// TIA Portal V17 export
// export: Created 2026-05-13T16:54:41.7855142Z, ExportSetting WithDefaults, DisplayName Totally Integrated Automation Portal, DisplayVersion V17 Update 4, DisplayName TIA Portal Openness, DisplayVersion V17 Update 4, DisplayName TIA Portal Version Control Interface, DisplayVersion V17, DisplayName SINAMICS Startdrive Advanced, DisplayVersion V17, DisplayName SINAMICS Startdrive G130, G150, S120, S150, SINAMICS MV, S210, DisplayVersion V17, DisplayName SINAMICS Startdrive G110M, G120, G120C, G120D, G120P, G115D, DisplayVersion V17, DisplayName STEP 7 Professional, DisplayVersion V17 Update 4, DisplayName STEP 7 Safety, DisplayVersion V17, DisplayName WinCC Professional, DisplayVersion V17 Update 4
TagTable "变量归档"
  进风温度 : Real  (1 s)
  出风温度 : Real  (1 s)
  data_id_1 : Int  (1 s)
  data_id_2 : Int  (1 s)
  data_id_3 : Int  (1 s)
  data_id_4 : Int  (1 s)
  data_id_5 : Int  (1 s)
  data_id_6 : Int  (1 s)
  data_id_7 : Int  (1 s)
  data_id_8 : Int  (1 s)
  data_id_9 : Int  (1 s)
  data_id_10 : Int  (1 s)
  data_id_11 : Int  (1 s)
  data_id_12 : Int  (1 s)
  data_id_13 : Int  (1 s)
  data_id_14 : Int  (1 s)
  data_id_15 : Int  (1 s)
  data_时间_1 : WString  (1 s)
  data_时间_2 : WString  (1 s)
  data_时间_3 : WString  (1 s)
  data_时间_4 : WString  (1 s)
  data_时间_5 : WString  (1 s)
  data_时间_6 : WString  (1 s)
  data_时间_7 : WString  (1 s)
  data_时间_8 : WString  (1 s)
  data_时间_9 : WString  (1 s)
  data_时间_10 : WString  (1 s)
  data_时间_11 : WString  (1 s)
  data_时间_12 : WString  (1 s)
  data_时间_13 : WString  (1 s)
  data_时间_14 : WString  (1 s)
  data_时间_15 : WString  (1 s)
  data_进风温度_1 : WString  (1 s)
  data_进风温度_2 : WString  (1 s)
  data_进风温度_3 : WString  (1 s)
  data_进风温度_4 : WString  (1 s)
  data_进风温度_5 : WString  (1 s)
  data_进风温度_6 : WString  (1 s)
  data_进风温度_7 : WString  (1 s)
  data_进风温度_8 : WString  (1 s)
  data_进风温度_9 : WString  (1 s)
  data_进风温度_10 : WString  (1 s)
  data_进风温度_11 : WString  (1 s)
  data_进风温度_12 : WString  (1 s)
  data_进风温度_13 : WString  (1 s)
  data_进风温度_14 : WString  (1 s)
  data_进风温度_15 : WString  (1 s)
  data_出风温度_1 : WString  (1 s)
  data_出风温度_2 : WString  (1 s)
  data_出风温度_3 : WString  (1 s)
  data_出风温度_4 : WString  (1 s)
  data_出风温度_5 : WString  (1 s)
  data_出风温度_6 : WString  (1 s)
  data_出风温度_7 : WString  (1 s)
  data_出风温度_8 : WString  (1 s)
  data_出风温度_9 : WString  (1 s)
  data_出风温度_10 : WString  (1 s)
  data_出风温度_11 : WString  (1 s)
  data_出风温度_12 : WString  (1 s)
  data_出风温度_13 : WString  (1 s)
  data_出风温度_14 : WString  (1 s)
  data_出风温度_15 : WString  (1 s)
  变量记录总页数 : Int  (1 s)
  变量记录当前页数 : Int  (1 s)
  data_执行说明 : WString  (1 s)
  开始时间 : DateTime  (1 s)
  结束时间 : DateTime  (1 s)
  启用时间段搜索 : Bool  (1 s)
  高效压差 : Real  (1 s)
  data_高效压差_1 : WString  (1 s)
  data_高效压差_2 : WString  (1 s)
  data_高效压差_3 : WString  (1 s)
  data_高效压差_4 : WString  (1 s)
  data_高效压差_5 : WString  (1 s)
  data_高效压差_6 : WString  (1 s)
  data_高效压差_7 : WString  (1 s)
  data_高效压差_8 : WString  (1 s)
  data_高效压差_9 : WString  (1 s)
  data_高效压差_10 : WString  (1 s)
  data_高效压差_11 : WString  (1 s)
  data_高效压差_12 : WString  (1 s)
  data_高效压差_13 : WString  (1 s)
  data_高效压差_14 : WString  (1 s)
  data_高效压差_15 : WString  (1 s)
  布袋压差 : Real  (1 s)
  data_布袋压差_1 : WString  (1 s)
  data_布袋压差_2 : WString  (1 s)
  data_布袋压差_3 : WString  (1 s)
  data_布袋压差_4 : WString  (1 s)
  data_布袋压差_5 : WString  (1 s)
  data_布袋压差_6 : WString  (1 s)
  data_布袋压差_7 : WString  (1 s)
  data_布袋压差_8 : WString  (1 s)
  data_布袋压差_9 : WString  (1 s)
  data_布袋压差_10 : WString  (1 s)
  data_布袋压差_11 : WString  (1 s)
  data_布袋压差_12 : WString  (1 s)
  data_布袋压差_13 : WString  (1 s)
  data_布袋压差_14 : WString  (1 s)
  data_布袋压差_15 : WString  (1 s)
  出口压差 : Real  (1 s)
  data_出口压差_1 : WString  (1 s)
  data_出口压差_2 : WString  (1 s)
  data_出口压差_3 : WString  (1 s)
  data_出口压差_4 : WString  (1 s)
  data_出口压差_5 : WString  (1 s)
  data_出口压差_6 : WString  (1 s)
  data_出口压差_7 : WString  (1 s)
  data_出口压差_8 : WString  (1 s)
  data_出口压差_9 : WString  (1 s)
  data_出口压差_10 : WString  (1 s)
  data_出口压差_11 : WString  (1 s)
  data_出口压差_12 : WString  (1 s)
  data_出口压差_13 : WString  (1 s)
  data_出口压差_14 : WString  (1 s)
  data_出口压差_15 : WString  (1 s)
  塔内压力 : Real  (1 s)
  data_塔内压力_1 : WString  (1 s)
  data_塔内压力_2 : WString  (1 s)
  data_塔内压力_3 : WString  (1 s)
  data_塔内压力_4 : WString  (1 s)
  data_塔内压力_5 : WString  (1 s)
  data_塔内压力_6 : WString  (1 s)
  data_塔内压力_7 : WString  (1 s)
  data_塔内压力_8 : WString  (1 s)
  data_塔内压力_9 : WString  (1 s)
  data_塔内压力_10 : WString  (1 s)
  data_塔内压力_11 : WString  (1 s)
  data_塔内压力_12 : WString  (1 s)
  data_塔内压力_13 : WString  (1 s)
  data_塔内压力_14 : WString  (1 s)
  data_塔内压力_15 : WString  (1 s)
  送风频率 : Real  (1 s)
  data_送风频率_1 : WString  (1 s)
  data_送风频率_2 : WString  (1 s)
  data_送风频率_3 : WString  (1 s)
  data_送风频率_4 : WString  (1 s)
  data_送风频率_5 : WString  (1 s)
  data_送风频率_6 : WString  (1 s)
  data_送风频率_7 : WString  (1 s)
  data_送风频率_8 : WString  (1 s)
  data_送风频率_9 : WString  (1 s)
  data_送风频率_10 : WString  (1 s)
  data_送风频率_11 : WString  (1 s)
  data_送风频率_12 : WString  (1 s)
  data_送风频率_13 : WString  (1 s)
  data_送风频率_14 : WString  (1 s)
  data_送风频率_15 : WString  (1 s)
  雾化频率 : Real  (1 s)
  data_雾化频率_1 : WString  (1 s)
  data_雾化频率_2 : WString  (1 s)
  data_雾化频率_3 : WString  (1 s)
  data_雾化频率_4 : WString  (1 s)
  data_雾化频率_5 : WString  (1 s)
  data_雾化频率_6 : WString  (1 s)
  data_雾化频率_7 : WString  (1 s)
  data_雾化频率_8 : WString  (1 s)
  data_雾化频率_9 : WString  (1 s)
  data_雾化频率_10 : WString  (1 s)
  data_雾化频率_11 : WString  (1 s)
  data_雾化频率_12 : WString  (1 s)
  data_雾化频率_13 : WString  (1 s)
  data_雾化频率_14 : WString  (1 s)
  data_雾化频率_15 : WString  (1 s)
  清洗压力 : Real  (1 s)
  data_清洗压力_1 : WString  (1 s)
  data_清洗压力_2 : WString  (1 s)
  data_清洗压力_3 : WString  (1 s)
  data_清洗压力_4 : WString  (1 s)
  data_清洗压力_5 : WString  (1 s)
  data_清洗压力_6 : WString  (1 s)
  data_清洗压力_7 : WString  (1 s)
  data_清洗压力_8 : WString  (1 s)
  data_清洗压力_9 : WString  (1 s)
  data_清洗压力_10 : WString  (1 s)
  data_清洗压力_11 : WString  (1 s)
  data_清洗压力_12 : WString  (1 s)
  data_清洗压力_13 : WString  (1 s)
  data_清洗压力_14 : WString  (1 s)
  data_清洗压力_15 : WString  (1 s)
  碱洗温度 : Real  (1 s)
  data_碱洗温度_1 : WString  (1 s)
  data_碱洗温度_2 : WString  (1 s)
  data_碱洗温度_3 : WString  (1 s)
  data_碱洗温度_4 : WString  (1 s)
  data_碱洗温度_5 : WString  (1 s)
  data_碱洗温度_6 : WString  (1 s)
  data_碱洗温度_7 : WString  (1 s)
  data_碱洗温度_8 : WString  (1 s)
  data_碱洗温度_9 : WString  (1 s)
  data_碱洗温度_10 : WString  (1 s)
  data_碱洗温度_11 : WString  (1 s)
  data_碱洗温度_12 : WString  (1 s)
  data_碱洗温度_13 : WString  (1 s)
  data_碱洗温度_14 : WString  (1 s)
  data_碱洗温度_15 : WString  (1 s)
  引风频率 : Real  (1 s)
  data_引风频率_1 : WString  (1 s)
  data_引风频率_2 : WString  (1 s)
  data_引风频率_3 : WString  (1 s)
  data_引风频率_4 : WString  (1 s)
  data_引风频率_5 : WString  (1 s)
  data_引风频率_6 : WString  (1 s)
  data_引风频率_7 : WString  (1 s)
  data_引风频率_8 : WString  (1 s)
  data_引风频率_9 : WString  (1 s)
  data_引风频率_10 : WString  (1 s)
  data_引风频率_11 : WString  (1 s)
  data_引风频率_12 : WString  (1 s)
  data_引风频率_13 : WString  (1 s)
  data_引风频率_14 : WString  (1 s)
  data_引风频率_15 : WString  (1 s)
  VBS_Run : Bool  (1 s)
  归记录开始 : Bool  (1 s)
  data_进风温度P_1 : WString  (1 s)
  data_进风温度P_2 : WString  (1 s)
  data_进风温度P_3 : WString  (1 s)
  data_进风温度P_4 : WString  (1 s)
  data_进风温度P_5 : WString  (1 s)
  data_进风温度P_6 : WString  (1 s)
  data_进风温度P_7 : WString  (1 s)
  data_进风温度P_8 : WString  (1 s)
  data_进风温度P_9 : WString  (1 s)
  data_进风温度P_10 : WString  (1 s)
  data_进风温度P_11 : WString  (1 s)
  data_进风温度P_12 : WString  (1 s)
  data_进风温度P_13 : WString  (1 s)
  data_进风温度P_14 : WString  (1 s)
  data_进风温度P_15 : WString  (1 s)
